(* CoDeSys 2.3.9.41 project: Armen_5_ред.pro *)
(* Libraries: Util.lib 18.5.10 15:14:28, STANDARD.LIB 4.10.05 11:14:46, IECSFC.LIB 13.4.06 15:51:28, SYSLIBTIME.LIB 20.2.06 12:31:16, SYSTASKINFO.LIB 20.2.06 12:31:38, ANALYZATION.LIB 5.10.99 09:05:06, SYSLIBCALLBACK.LIB 20.2.06 12:31:08, PID_Regulators.lib 28.12.06 16:47:54 *)

(* PLC configuration (modules and I/O channels)
Fast discrete inputs [I_SIMPLE_INPUT] node 0, in %IB0 out %QB0 {ChannellName = Fast discrete inputs; Filtrationtime = 10000}
  AT %IX0.0 [BitInput] Discrete input 1 {ChannellName = Enter name}
  AT %IX0.1 [BitInput] Discrete input 2 {ChannellName = Enter name}
AT %IB1.0 [ByteInput] 8 discrete inputs {ChannellName = Enter name}
AT %IB1.1 [ByteInput] 8 discrete inputs {ChannellName = Enter name}
Fan AT %QX2.0 [BitOutput] Fast discrete output 1 {ChannellName = Enter name}
Hot_fan AT %QX2.1 [BitOutput] Fast discrete output 2 {ChannellName = Enter name}
Fan_wall AT %QX2.2 [BitOutput] Fast discrete output 3 {ChannellName = Enter name}
Light_out AT %QX2.3 [BitOutput] Fast discrete output 4 {ChannellName = Enter name}
AT %QB3.0 [ByteOutput] 8 discrete outputs {ChannellName = Enter name}
AT %IX4.0 [BitInput] Special input {ChannellName = Enter name}
AT %QX5.0 [BitOutput] Special output {ChannellName = Enter name}
RS-232 [COM2_USART] node 0, in %IB6.0.0 out %QB6.0.0 {ChannellName = RS-232; CommunicationSpeed = 115200; Parity = NO PARITY CHECK; BitLength = 8 bits; StopLength = One stop bit; InterfaceType = RS232; FrameOriented = RTU; Timeout = 0; Visibility = No}
8 bits [8Bit] node 1, in %IB6.1 out %QB6.1 {ChannellName = 8 bit}
  AT %QB6.1.0 [ByteOutput] {ChannellName = Enter name}
8 bits [8Bit] node 2, in %IB6.2 out %QB6.2 {ChannellName = 8 bit}
  AT %QB6.2.0 [ByteOutput] {ChannellName = Enter name}
8 bits [8Bit] node 3, in %IB6.3 out %QB6.3 {ChannellName = 8 bit}
  AT %QB6.3.0 [ByteOutput] {ChannellName = Enter name}
8 bits [8Bit] node 4, in %IB6.4 out %QB6.4 {ChannellName = 8 bit}
  AT %QB6.4.0 [ByteOutput] {ChannellName = Enter name}
  AT %QB6.5.0 [ByteOutput] {ChannellName = Enter name}
  AT %QB6.6.0 [ByteOutput] {ChannellName = Enter name}
pH_i AT %QW6.7.0 [WordOutput] {ChannellName = Enter name}
EC_i AT %QW6.8.0 [WordOutput] {ChannellName = Enter name}
FanWall_t_start AT %QW6.9.0 [WordOutput] {ChannellName = Enter name}
FanWall_t_stop AT %QW6.10.0 [WordOutput] {ChannellName = Enter name}
Wind_set AT %QW6.11.0 [WordOutput] {ChannellName = Enter name}
Wind_Hyst AT %QW6.12.0 [WordOutput] {ChannellName = Enter name}
MODBUS_ID400Parameter.ChannellName1Modu AT %QW6.13.0 [WordOutput] e.Register2 byte2 byteSTRING2 byte / IB / %QB / %MB / %MFan_set {ChannellName = Enter name}
Fan_Hyst AT %QW6.14.0 [WordOutput] {ChannellName = Enter name}
MODBUS_ID400Parameter.ChannellName1Modu AT %QW6.15.0 [WordOutput] e.Register2 byte2 byteSTRING2 byteIB%QB%MB%MHot_set {ChannellName = Enter name}
Hot_Hyst AT %QW6.16.0 [WordOutput] {ChannellName = Enter name}
Cold_set AT %QW6.17.0 [WordOutput] {ChannellName = Enter name}
Cold_hyst AT %QW6.18.0 [WordOutput] {ChannellName = Enter name}
m_Light_on AT %QW6.19.0 [WordOutput] {ChannellName = Enter name}
h_light_on AT %QW6.20.0 [WordOutput] {ChannellName = Enter name}
m_light_off AT %QW6.21.0 [WordOutput] {ChannellName = Enter name}
h_light_off AT %QW6.22.0 [WordOutput] {ChannellName = Enter name}
MODBUS_ID400Parameter.ChannellName1Modu AT %QW6.23.0 [WordOutput] e.Register2 byte2 byteSTRING2 byteIB%QB%MB%Mt_tep_i {ChannellName = Enter name}
MODBUS_ID400Parameter.ChannellName1Modu AT %QW6.24.0 [WordOutput] e.Register2 byte2 byteSTRING2 byteIB%QB%MB%Mv_tep_i {ChannellName = Enter name}
t_ul_i AT %QW6.25.0 [WordOutput] {ChannellName = Enter name}
v_ul_i AT %QW6.26.0 [WordOutput] {ChannellName = Enter name}
ph AT %QW6.27.0 [WordOutput] {ChannellName = Enter name}
EC AT %QW6.28.0 [WordOutput] {ChannellName = Enter name}
AT %QW6.29.0 [WordOutput] {ChannellName = Enter name}
AT %QW6.30.0 [WordOutput] {ChannellName = Enter name}
AT %QW6.31.0 [WordOutput] {ChannellName = Enter name}
AT %QW6.32.0 [WordOutput] {ChannellName = Enter name}
AT %QW6.33.0 [WordOutput] {ChannellName = Enter name}
AT %QW6.34.0 [WordOutput] {ChannellName = Enter name}
AT %QW6.35.0 [WordOutput] {ChannellName = Enter name}
MODBUS_ID400Parameter.ChannellName1Modu AT %QW6.36.0 [WordOutput] e.Register2 byte2 byteSTRING2 byte$IB$%QB$%MB$%MH_panel {ChannellName = Enter name}
MODBUS_ID400Parameter.ChannellName1Modu AT %QW6.37.0 [WordOutput] e.Register2 byte2 byteSTRING2 byte%IB%%QB%%MB%%MM_panel {ChannellName = Enter name}
AT %QW6.38.0 [WordOutput] {ChannellName = Enter name}
AT %QW6.39.0 [WordOutput] {ChannellName = Enter name}
MODBUS_ID400Parameter.ChannellName1Modu AT %QW6.40.0 [WordOutput] e.Register2 byte2 byteSTRING2 byte(IB(%QB(%MB(%Mt_vod_i {ChannellName = Enter name}
Rash AT %QW6.41.0 [WordOutput] {ChannellName = Enter name}
P_i AT %QW6.42.0 [WordOutput] {ChannellName = Enter name}
Lvl_i AT %QW6.43.0 [WordOutput] {ChannellName = Enter name}
H_p1 AT %QW6.44.0 [WordOutput] {ChannellName = Enter name}
M_p1 AT %QW6.45.0 [WordOutput] {ChannellName = Enter name}
H_p2 AT %QW6.46.0 [WordOutput] {ChannellName = Enter name}
M_p2 AT %QW6.47.0 [WordOutput] {ChannellName = Enter name}
H_p3 AT %QW6.48.0 [WordOutput] {ChannellName = Enter name}
M_p3 AT %QW6.49.0 [WordOutput] {ChannellName = Enter name}
H_p4 AT %QW6.50.0 [WordOutput] {ChannellName = Enter name}
M_p4 AT %QW6.51.0 [WordOutput] {ChannellName = Enter name}
t_p1 AT %QW6.52.0 [WordOutput] {ChannellName = Enter name}
t_p2 AT %QW6.53.0 [WordOutput] {ChannellName = Enter name}
t_p3 AT %QW6.54.0 [WordOutput] {ChannellName = Enter name}
t_p4 AT %QW6.55.0 [WordOutput] {ChannellName = Enter name}
r_p1 AT %QW6.56.0 [WordOutput] {ChannellName = Enter name}
r_p2 AT %QW6.57.0 [WordOutput] {ChannellName = Enter name}
r_p3 AT %QW6.58.0 [WordOutput] {ChannellName = Enter name}
r_p4 AT %QW6.59.0 [WordOutput] {ChannellName = Enter name}
Pausa_p1 AT %QW6.60.0 [WordOutput] {ChannellName = Enter name}
Pausa_p2 AT %QW6.61.0 [WordOutput] {ChannellName = Enter name}
Pausa_p3 AT %QW6.62.0 [WordOutput] {ChannellName = Enter name}
Pausa_p4 AT %QW6.63.0 [WordOutput] {ChannellName = Enter name}
AT %QW6.64.0 [WordOutput] {ChannellName = Enter name}
AT %QD7.0 [DWordOutput] Last address {ChannellName = Enter name}
AT %QW7.1 [WordOutput] Last error {ChannellName = Enter name}
RS-485-1 [COM1_USART] node 0, in %IB7.0 out %QB7.0 {ChannellName = RS-485-1; CommunicationSpeed = 38400; Parity = NO PARITY CHECK; BitLength = 8 bits; StopLength = One stop bit; InterfaceType = RS485; FrameOriented = RTU; Timeout = 0; Visibility = No}
AT %QB7.1.0 [ComChannel] Command (0xff - Start) {ChannellName = Enter name}
Wind AT %QD7.1.0.0 [FloatOutput] {ChannellName = Enter name}
t_vod AT %QD7.1.1.0 [FloatOutput] {ChannellName = Enter name}
AT %QB7.2.0 [ComChannel] Command (0xff - Start) {ChannellName = Enter name}
t_tep AT %QW7.2.0.0 [WordOutput] {ChannellName = Enter name}
v_tep AT %QW7.2.1.0 [WordOutput] {ChannellName = Enter name}
AT %QB7.3.0 [ComChannel] Command (0xff - Start) {ChannellName = Enter name}
t_ul AT %QW7.3.0.0 [WordOutput] {ChannellName = Enter name}
v_ul AT %QW7.3.1.0 [WordOutput] {ChannellName = Enter name}
AT %QB7.4.0 [ComChannel] Command (0xff - Start) {ChannellName = Enter name}
PR100_in AT %QW7.4.0.0 [WordOutput] {ChannellName = Enter name}
PR100_out AT %QW7.4.1.0 [WordOutput] {ChannellName = Enter name}
ph_PR AT %QD7.4.2.0 [FloatOutput] {ChannellName = Enter name}
EC_PR AT %QD7.4.3.0 [FloatOutput] {ChannellName = Enter name}
p_PR AT %QD7.4.4.0 [FloatOutput] {ChannellName = Enter name}
*)

(* POU PLC_PRG, CFC *)
PROGRAM PLC_PRG
VAR
	Tof_Cold: TOF;
	FanWall: BLINK;
	Window_contr: HYSTERESIS;
	Hot_contr: HYSTERESIS;
	Cold_contr: HYSTERESIS;
	Tof_hot: TOF;

	Tof_wind: TOF;
	Window2_tim,Window2_tim_2: TON;
END_VAR
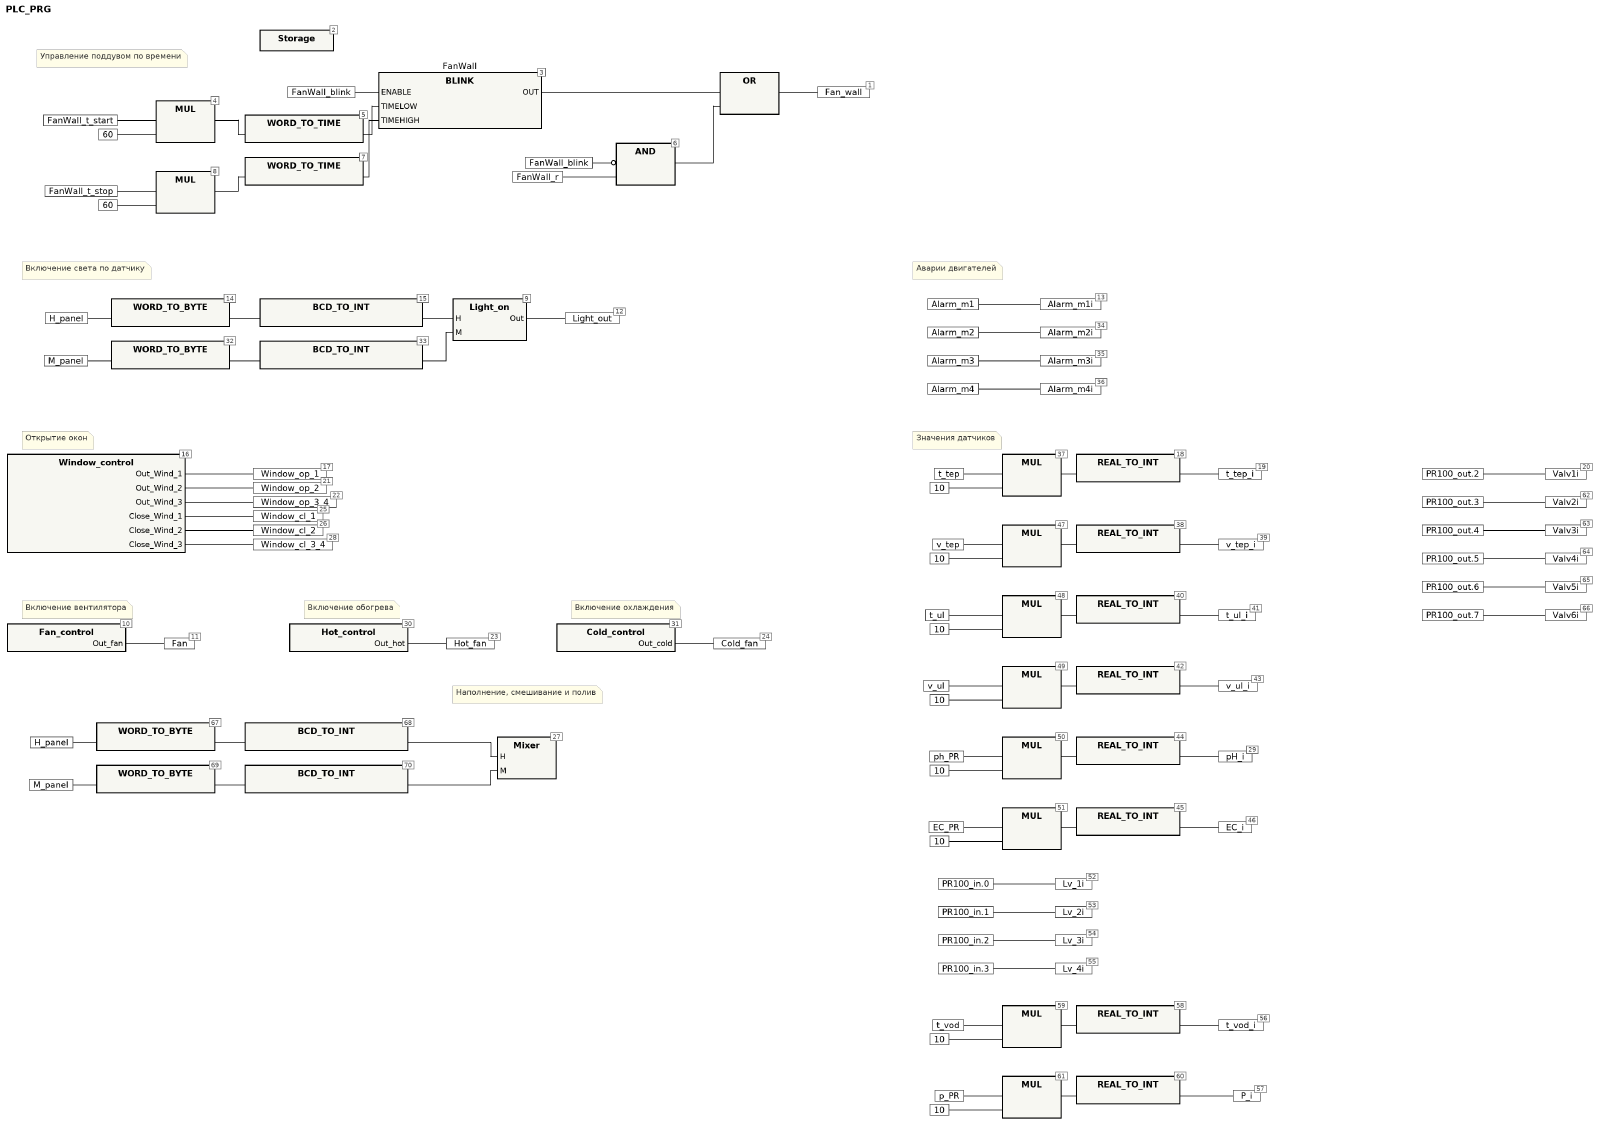
_CFC_ (* Continuous Function Chart, elements in execution order *)
(* Управление поддувом по времени *)
#0 OR(#3.OUT, #6)
#1 Fan_wall <= #0
#2 Storage()
#3 FanWall:BLINK(ENABLE: FanWall_blink, TIMELOW: #5, TIMEHIGH: #7)
#4 MUL(FanWall_t_start, 60)
#5 WORD_TO_TIME(#4)
#6 AND(NOT FanWall_blink, FanWall_r)
#7 WORD_TO_TIME(#8)
#8 MUL(FanWall_t_stop, 60)
(* Включение света по датчику *)
#9 Light_on(H: #15, M: #33)
#10 Fan_control()
#11 Fan <= #10.Out_fan
#12 Light_out <= #9.Out
#13 Alarm_m1i <= Alarm_m1
#14 WORD_TO_BYTE(H_panel)
#15 BCD_TO_INT(#14)
#16 Window_control()
#17 Window_op_1 <= #16.Out_Wind_1
#18 REAL_TO_INT(#37)
#19 t_tep_i <= #18
#20 Valv1i <= PR100_out.2
#21 Window_op_2 <= #16.Out_Wind_2
#22 Window_op_3_4 <= #16.Out_Wind_3
(* Открытие окон *)
(* Включение вентилятора *)
#23 Hot_fan <= #30.Out_hot
(* Включение обогрева *)
#24 Cold_fan <= #31.Out_cold
(* Включение охлаждения *)
#25 Window_cl_1 <= #16.Close_Wind_1
#26 Window_cl_2 <= #16.Close_Wind_2
#27 Mixer(H: #68, M: #70)
#28 Window_cl_3_4 <= #16.Close_Wind_3
#29 pH_i <= #44
#30 Hot_control()
#31 Cold_control()
(* Наполнение, смешивание и полив *)
#32 WORD_TO_BYTE(M_panel)
#33 BCD_TO_INT(#32)
(* Аварии двигателей *)
#34 Alarm_m2i <= Alarm_m2
#35 Alarm_m3i <= Alarm_m3
#36 Alarm_m4i <= Alarm_m4
(* Значения датчиков *)
#37 MUL(t_tep, 10)
#38 REAL_TO_INT(#47)
#39 v_tep_i <= #38
#40 REAL_TO_INT(#48)
#41 t_ul_i <= #40
#42 REAL_TO_INT(#49)
#43 v_ul_i <= #42
#44 REAL_TO_INT(#50)
#45 REAL_TO_INT(#51)
#46 EC_i <= #45
#47 MUL(v_tep, 10)
#48 MUL(t_ul, 10)
#49 MUL(v_ul, 10)
#50 MUL(ph_PR, 10)
#51 MUL(EC_PR, 10)
#52 Lv_1i <= PR100_in.0
#53 Lv_2i <= PR100_in.1
#54 Lv_3i <= PR100_in.2
#55 Lv_4i <= PR100_in.3
#56 t_vod_i <= #58
#57 P_i <= #60
#58 REAL_TO_INT(#59)
#59 MUL(t_vod, 10)
#60 REAL_TO_INT(#61)
#61 MUL(p_PR, 10)
#62 Valv2i <= PR100_out.3
#63 Valv3i <= PR100_out.4
#64 Valv4i <= PR100_out.5
#65 Valv5i <= PR100_out.6
#66 Valv6i <= PR100_out.7
#67 WORD_TO_BYTE(H_panel)
#68 BCD_TO_INT(#67)
#69 WORD_TO_BYTE(M_panel)
#70 BCD_TO_INT(#69)
_END_CFC_
END_PROGRAM

(* POU Storage, ST *)
PROGRAM Storage
VAR
	flag:BOOL;
END_VAR

VAR RETAIN
	mas1: ARRAY [1..100] OF BOOL;
	mas2: ARRAY [1..50] OF WORD;
END_VAR
	IF flag=0 THEN

(************* wORD ***********)
	pH_i:=mas2[1];
	EC_i:=mas2[2];
	FanWall_t_start:=mas2[3];
	FanWall_t_stop:=mas2[4];
	Wind_set:=mas2[5];
	Wind_Hyst:=mas2[6];
	Fan_set:=mas2[7];
	Fan_Hyst:=mas2[8];
	Hot_set:=mas2[9];
	Hot_Hyst:=mas2[10];
	Cold_set:=mas2[11];
	Cold_hyst:=mas2[12];
	m_Light_on:=mas2[13];
	h_light_on:=mas2[14];
	m_light_off:=mas2[15];
	h_light_off:=mas2[16];
	ph:=mas2[17];
	EC:=mas2[18];
	Rash:=mas2[19];

	H_p1:=mas2[20];
	M_p1:=mas2[21];
	H_p2:=mas2[22];
	M_p2:=mas2[23];
	H_p3:=mas2[24];
	M_p3:=mas2[25];
	H_p4:=mas2[26];
	M_p4:=mas2[27];
	t_p1:=mas2[28];
	t_p2:=mas2[29];
	t_p3:=mas2[30];
	t_p4:=mas2[31];
	r_p1:=mas2[32];
	r_p2:=mas2[33];
	r_p3:=mas2[34];
	r_p4:=mas2[35];
	Pausa_p1:=mas2[36];
	Pausa_p2:=mas2[37];
	Pausa_p3:=mas2[38];
	Pausa_p4:=mas2[39];

	flag:=1;

		IF Wind_set=0 THEN   (*** Проверка значений при первом пуске ***)
			FanWall_t_start:=15;
			FanWall_t_stop:=15;
			Wind_set:=200;
			Wind_Hyst:=10;
			Fan_set:=200;
			Fan_Hyst:=10;
			Hot_set:=200;
			Hot_Hyst:=10;
			Cold_set:=200;
			Cold_hyst:=10;
			h_light_on:=23;
			h_light_off:=5;
			r_p1:=1;
			r_p2:=1;
			r_p3:=1;
			r_p4:=1;

		END_IF;

	ELSE


(************* wORD ***********)
	mas2[1]:=pH_i;
	mas2[2]:=EC_i;
	mas2[3]:=FanWall_t_start;
	mas2[4]:=FanWall_t_stop;
	mas2[5]:=Wind_set;
	mas2[6]:=Wind_Hyst;
	mas2[7]:=Fan_set;
	mas2[8]:=Fan_Hyst;
	mas2[9]:=Hot_set;
	mas2[10]:=Hot_Hyst;
	mas2[11]:=Cold_set;
	mas2[12]:=Cold_hyst;
	mas2[13]:=m_Light_on;
	mas2[14]:=h_light_on;
	mas2[15]:=m_light_off;
	mas2[16]:=h_light_off;
	mas2[17]:=ph;
	mas2[18]:=EC;
	mas2[19]:=Rash;

	mas2[20]:=H_p1;
	mas2[21]:=M_p1;
	mas2[22]:=H_p2;
	mas2[23]:=M_p2;
	mas2[24]:=H_p3;
	mas2[25]:=M_p3;
	mas2[26]:=H_p4;
	mas2[27]:=M_p4;
	mas2[28]:=t_p1;
	mas2[29]:=t_p2;
	mas2[30]:=t_p3;
	mas2[31]:=t_p4;
	mas2[32]:=r_p1;
	mas2[33]:=r_p2;
	mas2[34]:=r_p3;
	mas2[35]:=r_p4;
	mas2[36]:=Pausa_p1;
	mas2[37]:=Pausa_p2;
	mas2[38]:=Pausa_p3;
	mas2[39]:=Pausa_p4;


	END_IF
END_PROGRAM

(* POU Light_on, ST *)
PROGRAM Light_on
VAR
END_VAR
VAR_OUTPUT
	Out: BOOL;
END_VAR
VAR_INPUT
	H, M: INT;
END_VAR
IF Light_auto=1 THEN
	IF Light_str_sensor=1 THEN
		Out:=Light_str_sensor;
	END_IF

	IF (Light_str_sensor=0) THEN
		IF ((m_Light_on+h_Light_on*100)<(M+H*100)) OR ( (m_Light_off+h_Light_off*100)>(M+H*100)) THEN
			Out:=1;
		ELSE
			Out:=0;
		END_IF
	END_IF

	Light_r:=0;
ELSE
	Light_str_sensor:=0;
	Out:=Light_r;
END_IF

(*Сброс для вентилятора наддува*)

	IF FanWall_blink =1 THEN
		FanWall_r:=0;
	END_IF
END_PROGRAM

(* POU Fan_control, ST *)
PROGRAM Fan_control
VAR
	Hyst: HYSTERESIS;
	T1: TOF;
END_VAR
VAR_OUTPUT
	Out_fan: BOOL;
END_VAR
IF Fan_auto=1 THEN
T1(PT:= T#20s);
Hyst(IN:=REAL_TO_INT(t_tep) *10*(-1));
Hyst.HIGH:= WORD_TO_INT(Fan_set+Fan_Hyst/2)*(-1);
Hyst.low:=WORD_TO_INT( Fan_set-Fan_Hyst/2)*(-1);

	IF Hyst.OUT AND (NOT(t1.Q )) THEN
		Out_fan:=1;
		T1.IN:=1;
	END_IF

	IF NOT(Hyst.OUT) AND T1.Q THEN
		Out_fan:=0;
		T1.IN:=0;
	END_IF

	Fan_r:=0;
ELSE
	Out_fan:=Fan_r;
END_IF
END_PROGRAM

(* POU Window_control, ST *)
PROGRAM Window_control
VAR
	Hyst: HYSTERESIS;
	 flag, flag2: BOOL;
	T1, Tw_op: TON;
END_VAR
VAR_OUTPUT
	Out_Wind_1, Out_Wind_2, Out_Wind_3: BOOL;
	Close_Wind_1, Close_Wind_2, Close_Wind_3: BOOL;
END_VAR
IF Wind_auto=1 THEN
T1(PT:= T#20s);
Tw_op(PT:= T#20s);
Hyst(IN:=REAL_TO_INT(t_tep) *10*(-1));
Hyst.HIGH:= WORD_TO_INT(Wind_set+Wind_Hyst/2)*(-1);
Hyst.low:=WORD_TO_INT(Wind_set-Wind_Hyst/2)*(-1);

	IF flag=0 THEN
		IF Hyst.OUT=1 THEN
			flag:=1;
		END_IF
	ELSE
		IF Hyst.OUT=0 THEN
			flag2:=1;
		END_IF
	END_IF

	IF wind>50 THEN
		flag2:=1;
	END_IF


	IF flag2=1 THEN
		flag:=NOT T1.Q; (*Сброс таймеров*)
		flag2:=NOT T1.Q;

	END_IF

	T1.IN:=flag2;

	Tw_op.IN:=Hyst.OUT AND (NOT flag2);

	(*Этапы открытия окон*)

	IF Tw_op.ET<t#10s THEN
		Out_Wind_1:=1;
		Out_Wind_2:=1;
		Out_Wind_3:=0;
	END_IF

	IF (Tw_op.ET>t#10s) AND (Tw_op.ET<t#20s) THEN
		Out_Wind_1:=0;
		Out_Wind_2:=0;
		Out_Wind_3:=1;
	END_IF

	IF ((Hyst.OUT AND (NOT flag2))=FALSE) OR Tw_op.Q THEN
		Out_Wind_1:=0;
		Out_Wind_2:=0;
		Out_Wind_3:=0;
	END_IF

(*Этапы закрытия окон*)

	IF T1.ET<t#10s AND flag2 THEN
		Close_Wind_1:=1;
		Close_Wind_2:=1;
		Close_Wind_3:=0;
	END_IF

	IF (T1.ET>t#10s) AND (T1.ET<t#20s) THEN
		Close_Wind_1:=0;
		Close_Wind_2:=0;
		Close_Wind_3:=1;
	END_IF

	IF (Hyst.OUT =TRUE) OR T1.Q THEN
		Close_Wind_1:=0;
		Close_Wind_2:=0;
		Close_Wind_3:=0;
	END_IF

	IF (Out_Wind_1=1) OR (Out_Wind_2=1) OR ( Out_Wind_3=1) THEN
		Close_Wind_1:=0;
		Close_Wind_2:=0;
		Close_Wind_3:=0;
	END_IF
	(*Сброс ручных настроек*)
	Wind_r1:=0;
	Wind_r2:=0;
	Wind_r3_4:=0;
	Wind_r1_cl:=0;
	Wind_r2_cl:=0;
	Wind_r3_4_cl:=0;

ELSE	(*Ручное управление*)
	Out_Wind_1:=Wind_r1;
	Out_Wind_2:=Wind_r2;
	Out_Wind_3:=Wind_r3_4;
	Close_Wind_1:=Wind_r1_cl;
	Close_Wind_2:=Wind_r2_cl;
	Close_Wind_3:=	Wind_r3_4_cl;
	IF Wind_r1 AND Window_cl_1 THEN
		Wind_r1_cl:=0;
	END_IF
	IF Wind_r2 AND Window_cl_2 THEN
		Wind_r2_cl:=0;
	END_IF
	IF Window_op_3_4 AND Wind_r3_4_cl THEN
		Wind_r3_4_cl:=0;
	END_IF

	 flag:=0;
	 flag2:=0;

END_IF
END_PROGRAM

(* POU Mixer, ST *)
PROGRAM Mixer
	VAR RETAIN
	flag, f_b, f_m,p1,p2,p3,p4, f_res: BOOL;
	CT,CT1:CTU;
	T:BLINK;
	p1_off, p2_off, p3_off, p4_off: WORD; (*** Время окончания поливов ***)
END_VAR

VAR_INPUT
	H,M: INT;
END_VAR
	IF Auto_water=0 THEN
		PR100_out.0:=Pump;
		PR100_out.2:=Valv1;
		PR100_out.3:=Valv2;
		PR100_out.4:=Valv3;
		PR100_out.5:=Valv4;
		PR100_out.6:=Valv5;
		PR100_out.7:=Valv6;
		flag:=0;
	ELSE
		IF flag=0 THEN  (*Обнуление выходных сигналов *)
			PR100_out.0:=0;
			PR100_out.2:=0;
			PR100_out.3:=0;
			PR100_out.4:=0;
			PR100_out.5:=0;
			PR100_out.6:=0;
			PR100_out.7:=0;
			flag:=1;
		END_IF
	END_IF

 (*Наполнение емкости*)
	IF  (Auto_water=1) THEN
		IF (PR100_in.0=1) AND (f_b=0)  THEN
			f_b:=1;
			PR100_out.2:=0;
			CT.RESET:=1; (*сброс счётчика*)
			CT1.CU:=0;
			PR100_out.3:=1;
			PR100_out.4:=1;
			PR100_out.5:=1;
		ELSE
			PR100_out.2:=1;
		END_IF


	END_IF

(*Смешивание*)
	IF (f_b=1) AND (f_m=0) AND (Auto_water=1) THEN
		IF ph>=ph_PR THEN
			PR100_out.3:=0;
			PR100_out.4:=0;
		END_IF
		IF ec>=ec_PR THEN
			PR100_out.5:=0;
		END_IF
		f_m:=(fa AND fc) OR (NOT(PR100_in.4));
		PR100_out.6:=NOT(f_m);
		PR100_out.0:=(NOT(f_m)); (*защита от сухого хода*)
	END_IF
(*Полив*)

	IF (f_b=1) AND (f_m=1) AND (Auto_water=1) AND (CT1.Q=FALSE) AND ((pr1 OR pr2 OR pr3 OR pr4)=TRUE) AND (T.OUT=TRUE) THEN
		IF PR100_in.1=1 THEN		(*Условие работы до 3-го датчика уровня*)
			PR100_out.0:=TRUE AND PR100_out.1;
			PR100_out.7:=1;
		ELSE
			PR100_out.0:=0;
			PR100_out.7:=0;
			f_b:=0;
			f_m:=0;
			fc:=0;
			fa:=0;
			CT1.CU:=1;
		END_IF

		CT(pv:=9000);
		ct.CU:=Rashod;

	END_IF


	PR100_out.1:=PR100_in.3 AND PR100_out.0;(*защита от сухого хода*)
	Rash:=ct.CV*10;

(*** Условия полива ***)

(*** Исключение пересечений ***)
	IF H_p1>=H_p2 THEN
		IF (H_p2+1)<>24 THEN
			H_p2:=H_p2+1;
		ELSE
			H_p1:=H_p1-1;
		END_IF
	END_IF

	IF H_p2>=H_p3 THEN
		IF (H_p3+1)<>24 THEN
			H_p3:=H_p3+1;
		ELSE
			H_p2:=H_p2-1;
		END_IF
	END_IF

	IF H_p3>=H_p4 THEN
		IF (H_p4+1)<>24 THEN
			H_p4:=H_p4+1;
		ELSE
			H_p3:=H_p3-1;
		END_IF
	END_IF

	IF  ((M+H*100) = (H_p1*100+M_p1)) AND (pr1=1) THEN 	(* Определение полива *)
		IF p1=0 THEN
			CT1.RESET:=1;
			CT1.RESET:=0;
		END_IF
			CT1(pv:=r_p1);
			T.TIMEHIGH:=WORD_TO_TIME(t_p1*60);
			T.TIMELOW:=WORD_TO_TIME(Pausa_p1*60);
			p1:=1;
			p2:=0;
			p3:=0;
			p4:=0;
	END_IF

	IF  ((M+H*100) = (H_p2*100+M_p2))  AND (pr2=1) THEN 	(* Определение полива *)
		IF p2=0 THEN
			CT1.RESET:=1;
			CT1.RESET:=0;
		END_IF
			CT1(pv:=r_p2);
			T.TIMEHIGH:=WORD_TO_TIME(t_p2*60);
			T.TIMELOW:=WORD_TO_TIME(Pausa_p2*60);
			p1:=0;
			p2:=1;
			p3:=0;
			p4:=0;
	END_IF


	IF  ((M+H*100) = (H_p3*100+M_p3))  AND (pr3=1) THEN 	(* Определение полива *)
		IF p3=0 THEN
			CT1.RESET:=1;
			CT1.RESET:=0;
		END_IF
			CT1(pv:=r_p3);
			T.TIMEHIGH:=WORD_TO_TIME(t_p3*60);
			T.TIMELOW:=WORD_TO_TIME(Pausa_p3*60);
			p1:=0;
			p2:=0;
			p3:=1;
			p4:=0;
	END_IF


	IF  ((M+H*100) = (H_p4*100+M_p4))  AND (pr4=1) THEN 	(* Определение полива *)
		IF p4=0 THEN
			CT1.RESET:=1;
			CT1.RESET:=0;
		END_IF
			CT1(pv:=r_p4);
			T.TIMEHIGH:=WORD_TO_TIME(t_p4*60);
			T.TIMELOW:=WORD_TO_TIME(Pausa_p4*60);
			p1:=0;
			p2:=0;
			p3:=0;
			p4:=1;
	END_IF

	T(ENABLE:=NOT(CT1.Q) AND (pr1 OR pr2 OR pr3 OR pr4));

	(* Суточный сброс счётчиков *)

	IF (h+m) =0 THEN
		f_res:=1;
	END_IF

	IF (f_res=1) AND (CT1.Q=1) THEN
		f_res:=0;
		CT1(RESET:=1);
		CT1.RESET:=0;
	END_IF
END_PROGRAM

(* POU Hot_control, ST *)
PROGRAM Hot_control
VAR
	Hyst: HYSTERESIS;
	 flag, flag2: BOOL;
	T1: TON;
END_VAR
VAR_OUTPUT
	Out_hot: BOOL;
END_VAR
IF Hot_auto=1 THEN
T1(PT:= T#20s);
Hyst(IN:=REAL_TO_INT(t_tep) *10);
Hyst.HIGH:= Hot_set+Hot_Hyst/2;
Hyst.low:= Hot_set-Hot_Hyst/2;

	IF Hyst.OUT AND (NOT(t1.Q )) THEN
		Out_hot:=1;
		T1.IN:=1;
	END_IF

	IF NOT(Hyst.OUT) AND T1.Q THEN
		Out_hot:=0;
		T1.IN:=0;
	END_IF

	Hot_r:=0;
ELSE
	Out_hot:=Hot_r;
END_IF
END_PROGRAM

(* POU Cold_control, ST *)
PROGRAM Cold_control
VAR
	Hyst: HYSTERESIS;
	T1: TOF;
END_VAR
VAR_OUTPUT
	Out_cold: BOOL;
END_VAR
IF Cold_auto=1 THEN
	T1(PT:= T#20s);
	Hyst(IN:=REAL_TO_INT(t_tep) *10*(-1));
	Hyst.HIGH:= WORD_TO_INT(Cold_set+Cold_hyst/2)*(-1);
	Hyst.low:= WORD_TO_INT(Cold_set-Cold_hyst/2)*(-1);

	IF Hyst.OUT AND (NOT(t1.Q )) THEN
		Out_cold:=1;
		T1.IN:=1;
	END_IF

	IF NOT(Hyst.OUT) AND T1.Q THEN
		Out_cold:=0;
		T1.IN:=0;
	END_IF

	Cold_r:=0;
ELSE
	Out_cold:=Cold_r;
END_IF
END_PROGRAM
